FUNCTION_BLOCK MQTTPUBLISH_73D9883955B65591 (* Generic Interface Function Block Type *)
  (* Standard: 61499-2 *)
  (* Version 0.0, 05/11/2020, SESA489471, nxtControl GmBH, Template *)
  PACKAGE UAO.Hackathon;
  (* Compiler Cpp nxtControl builtin 1.0 *)
  {SET_ATTRIBUTE(Runtime.FBType.ImplementingType, nxtControl.CommProtocols#DYNGEN_MQTTPUBLISH)}
  {SET_ATTRIBUTE(Configuration.GenericFBType.InterfaceParams, nxtControl.CommProtocols#CNTX:=1)}
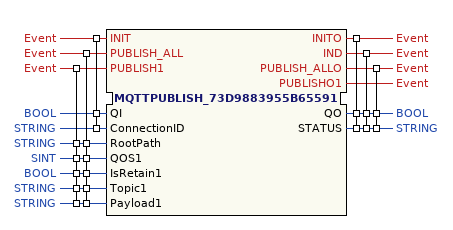
  EVENT_INPUT
    INIT WITH QI, ConnectionID; (* Request events for dedicated input data sets *)
    PUBLISH_ALL WITH Topic1, Payload1, RootPath, IsRetain1, QOS1;
    PUBLISH1 WITH Topic1, Payload1, RootPath, IsRetain1, QOS1;
  END_EVENT
  EVENT_OUTPUT
    INITO WITH QO, STATUS; (* Confirmation from Resource for a dedicated request *)
    IND WITH STATUS, QO;
    PUBLISH_ALLO WITH QO, STATUS; (* Indication from Resource *)
    PUBLISHO1;
  END_EVENT
  VAR_INPUT
    QI : BOOL;
    ConnectionID : STRING;
    RootPath : STRING;
    QOS1 : SINT;
    IsRetain1 : BOOL;
    Topic1 : STRING;
    Payload1 : STRING;
  END_VAR
  VAR_OUTPUT
    QO : BOOL; (* Input data from resource *)
    STATUS : STRING;
  END_VAR
  EC_STATES
    START;
  END_STATES
END_FUNCTION_BLOCK
